// Slaapkamer 1 bed R B11L00
TYPE ST_WP_Bedroom1BedR :
STRUCT
	fbButton1		: FB_DigitalIn;
	fbButton2		: FB_DigitalIn;
END_STRUCT
END_TYPE

(* stored: Version 1.1.0.1, ProductVersion 3.1.4024.12
   DUT ST_WP_Bedroom1BedR: Id {cbf36940-9b94-4cd7-9716-ef33fbcb17f3} *)
